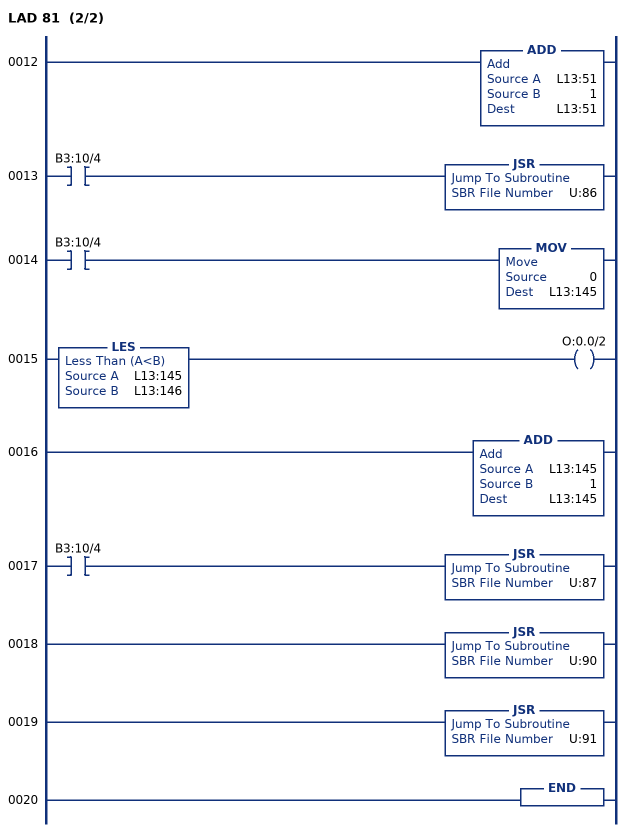
% Rung: 12 %
SOR ADD L13:51 1 L13:51 EOR
% Rung: 13 %
SOR XIC B3:10/4 JSR U:86 EOR
% Rung: 14 %
SOR XIC B3:10/4 MOV 0 L13:145 EOR
% Rung: 15 %
SOR LES L13:145 L13:146 OTE O:0.0/2 EOR
% Rung: 16 %
SOR ADD L13:145 1 L13:145 EOR
% Rung: 17 %
SOR XIC B3:10/4 JSR U:87 EOR
% Rung: 18 %
SOR JSR U:90 EOR
% Rung: 19 %
SOR JSR U:91 EOR
% Rung: 20 %
SOR END EOR

LADDER 82
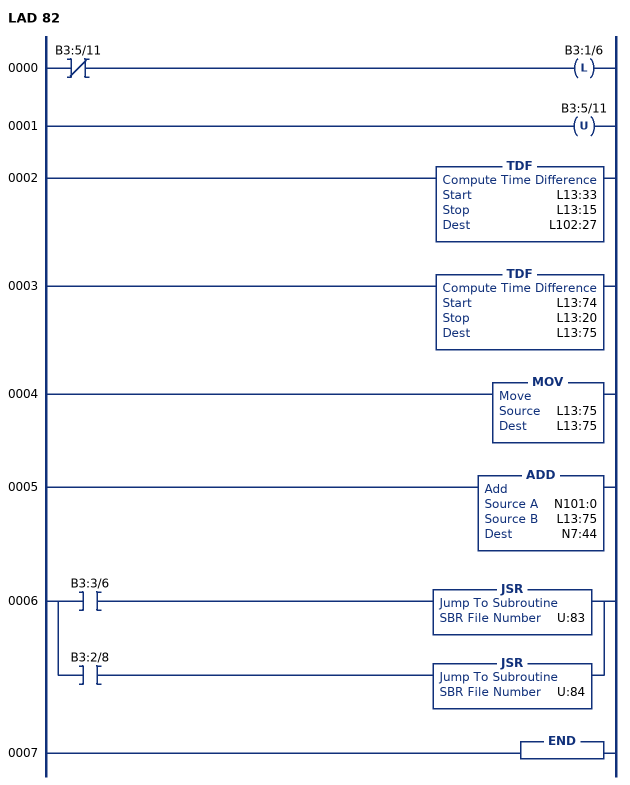
% Rung: 0 %
SOR XIO B3:5/11 OTL B3:1/6 EOR
% Rung: 1 %
SOR OTU B3:5/11 EOR
% Rung: 2 %
SOR TDF L13:33 L13:15 L102:27 EOR
% Rung: 3 %
SOR TDF L13:74 L13:20 L13:75 EOR
% Rung: 4 %
SOR MOV L13:75 L13:75 EOR
% Rung: 5 %
SOR ADD N101:0 L13:75 N7:44 EOR
% Rung: 6 %
SOR BST XIC B3:3/6 JSR U:83 NXB XIC B3:2/8 JSR U:84 BND EOR
% Rung: 7 %
SOR END EOR

LADDER 83
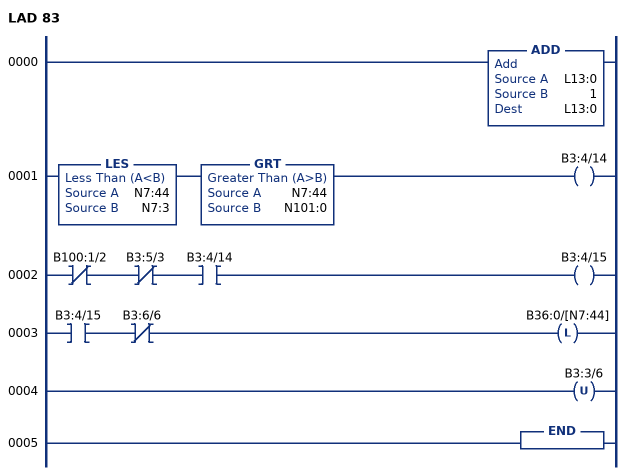
% Rung: 0 %
SOR ADD L13:0 1 L13:0 EOR
% Rung: 1 %
SOR LES N7:44 N7:3 GRT N7:44 N101:0 OTE B3:4/14 EOR
% Rung: 2 %
SOR XIO B100:1/2 XIO B3:5/3 XIC B3:4/14 OTE B3:4/15 EOR
% Rung: 3 %
SOR XIC B3:4/15 XIO B3:6/6 OTL B36:0/[N7:44] EOR
% Rung: 4 %
SOR OTU B3:3/6 EOR
% Rung: 5 %
SOR END EOR

LADDER 84
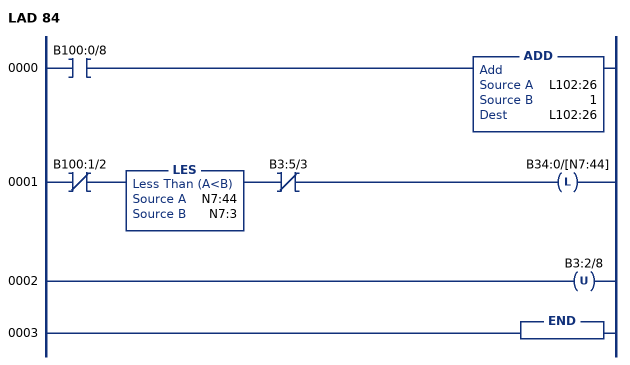
% Rung: 0 %
SOR XIC B100:0/8 ADD L102:26 1 L102:26 EOR
% Rung: 1 %
SOR XIO B100:1/2 LES N7:44 N7:3 XIO B3:5/3 OTL B34:0/[N7:44] EOR
% Rung: 2 %
SOR OTU B3:2/8 EOR
% Rung: 3 %
SOR END EOR

LADDER 85
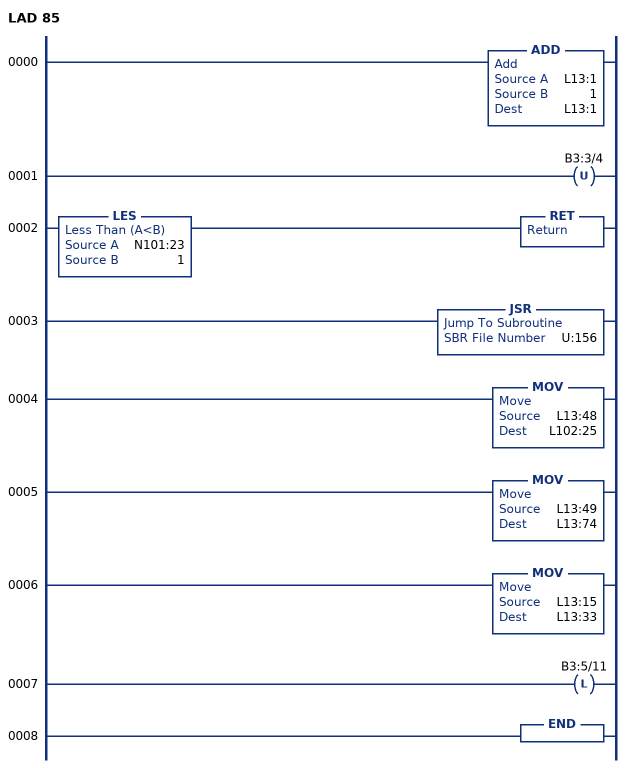
% Rung: 0 %
SOR ADD L13:1 1 L13:1 EOR
% Rung: 1 %
SOR OTU B3:3/4 EOR
% Rung: 2 %
SOR LES N101:23 1 RET EOR
% Rung: 3 %
SOR JSR U:156 EOR
% Rung: 4 %
SOR MOV L13:48 L102:25 EOR
% Rung: 5 %
SOR MOV L13:49 L13:74 EOR
% Rung: 6 %
SOR MOV L13:15 L13:33 EOR
% Rung: 7 %
SOR OTL B3:5/11 EOR
% Rung: 8 %
SOR END EOR

LADDER 86
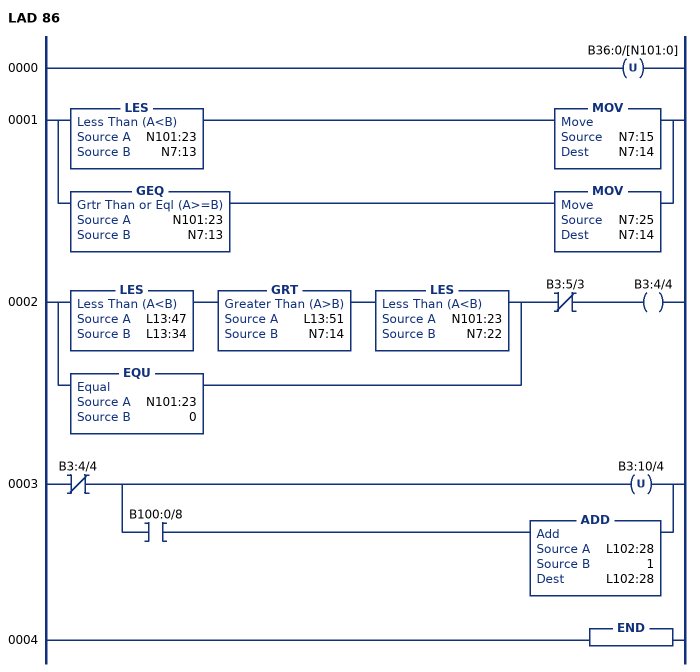
% Rung: 0 %
SOR OTU B36:0/[N101:0] EOR
% Rung: 1 %
SOR BST LES N101:23 N7:13 MOV N7:15 N7:14 NXB GEQ N101:23 N7:13 MOV N7:25 N7:14 BND EOR
% Rung: 2 %
SOR BST LES L13:47 L13:34 GRT L13:51 N7:14 LES N101:23 N7:22 NXB EQU N101:23 0 BND XIO B3:5/3 OTE B3:4/4 EOR
% Rung: 3 %
SOR XIO B3:4/4 BST OTU B3:10/4 NXB XIC B100:0/8 ADD L102:28 1 L102:28 BND EOR
% Rung: 4 %
SOR END EOR

LADDER 87
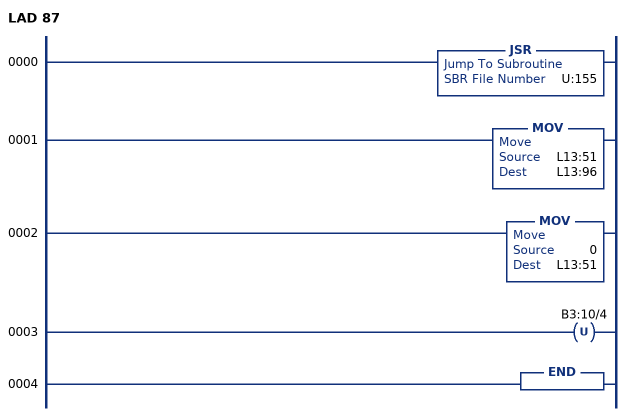
% Rung: 0 %
SOR JSR U:155 EOR
% Rung: 1 %
SOR MOV L13:51 L13:96 EOR
% Rung: 2 %
SOR MOV 0 L13:51 EOR
% Rung: 3 %
SOR OTU B3:10/4 EOR
% Rung: 4 %
SOR END EOR

LADDER 90
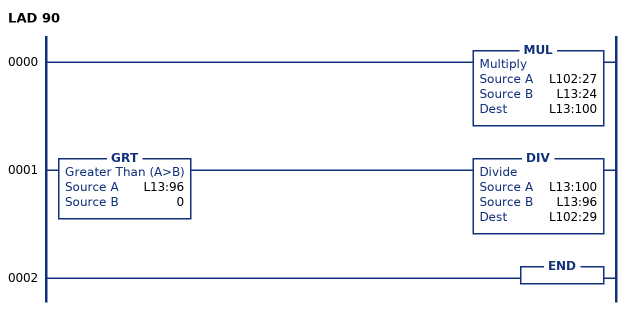
% Rung: 0 %
SOR MUL L102:27 L13:24 L13:100 EOR
% Rung: 1 %
SOR GRT L13:96 0 DIV L13:100 L13:96 L102:29 EOR
% Rung: 2 %
SOR END EOR

LADDER 91
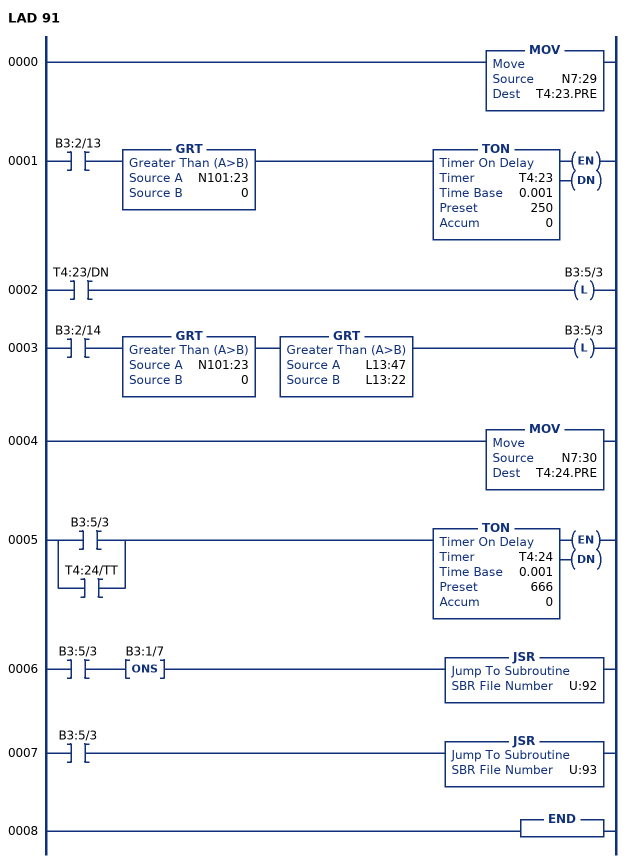
% Rung: 0 %
SOR MOV N7:29 T4:23.PRE EOR
% Rung: 1 %
SOR XIC B3:2/13 GRT N101:23 0 TON T4:23 0.001 250 0 EOR
% Rung: 2 %
SOR XIC T4:23/DN OTL B3:5/3 EOR
% Rung: 3 %
SOR XIC B3:2/14 GRT N101:23 0 GRT L13:47 L13:22 OTL B3:5/3 EOR
% Rung: 4 %
SOR MOV N7:30 T4:24.PRE EOR
% Rung: 5 %
SOR BST XIC B3:5/3 NXB XIC T4:24/TT BND TON T4:24 0.001 666 0 EOR
% Rung: 6 %
SOR XIC B3:5/3 ONS B3:1/7 JSR U:92 EOR
% Rung: 7 %
SOR XIC B3:5/3 JSR U:93 EOR
% Rung: 8 %
SOR END EOR

LADDER 92
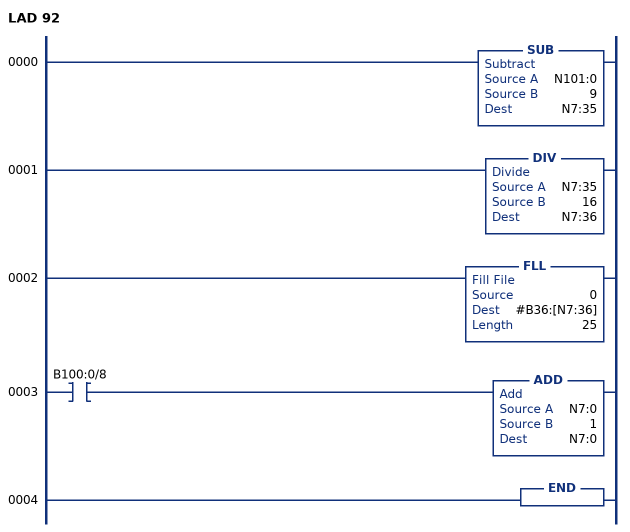
% Rung: 0 %
SOR SUB N101:0 9 N7:35 EOR
% Rung: 1 %
SOR DIV N7:35 16 N7:36 EOR
% Rung: 2 %
SOR FLL 0 #B36:[N7:36] 25 EOR
% Rung: 3 %
SOR XIC B100:0/8 ADD N7:0 1 N7:0 EOR
% Rung: 4 %
SOR END EOR

LADDER 93
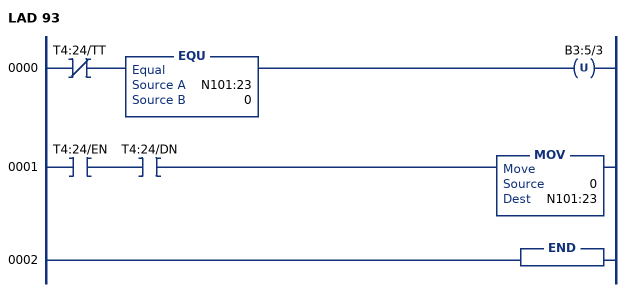
% Rung: 0 %
SOR XIO T4:24/TT EQU N101:23 0 OTU B3:5/3 EOR
% Rung: 1 %
SOR XIC T4:24/EN XIC T4:24/DN MOV 0 N101:23 EOR
% Rung: 2 %
SOR END EOR

LADDER 135
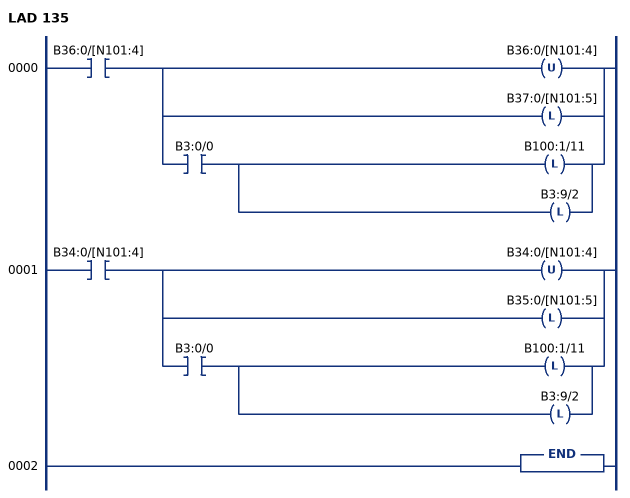
% Rung: 0 %
SOR XIC B36:0/[N101:4] BST OTU B36:0/[N101:4] NXB OTL B37:0/[N101:5] NXB XIC B3:0/0 BST OTL B100:1/11 NXB OTL B3:9/2 BND BND EOR
% Rung: 1 %
SOR XIC B34:0/[N101:4] BST OTU B34:0/[N101:4] NXB OTL B35:0/[N101:5] NXB XIC B3:0/0 BST OTL B100:1/11 NXB OTL B3:9/2 BND BND EOR
% Rung: 2 %
SOR END EOR

LADDER 137
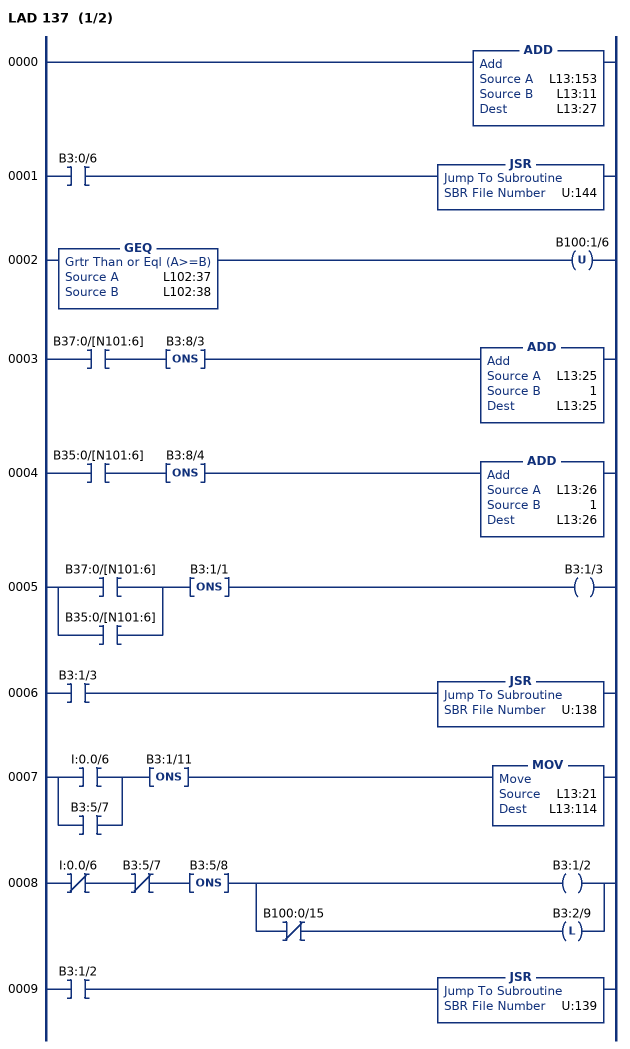
% Rung: 0 %
SOR ADD L13:153 L13:11 L13:27 EOR
% Rung: 1 %
SOR XIC B3:0/6 JSR U:144 EOR
% Rung: 2 %
SOR GEQ L102:37 L102:38 OTU B100:1/6 EOR
% Rung: 3 %
SOR XIC B37:0/[N101:6] ONS B3:8/3 ADD L13:25 1 L13:25 EOR
% Rung: 4 %
SOR XIC B35:0/[N101:6] ONS B3:8/4 ADD L13:26 1 L13:26 EOR
% Rung: 5 %
SOR BST XIC B37:0/[N101:6] NXB XIC B35:0/[N101:6] BND ONS B3:1/1 OTE B3:1/3 EOR
% Rung: 6 %
SOR XIC B3:1/3 JSR U:138 EOR
% Rung: 7 %
SOR BST XIC I:0.0/6 NXB XIC B3:5/7 BND ONS B3:1/11 MOV L13:21 L13:114 EOR
% Rung: 8 %
SOR XIO I:0.0/6 XIO B3:5/7 ONS B3:5/8 BST OTE B3:1/2 NXB XIO B100:0/15 OTL B3:2/9 BND EOR
% Rung: 9 %
SOR XIC B3:1/2 JSR U:139 EOR

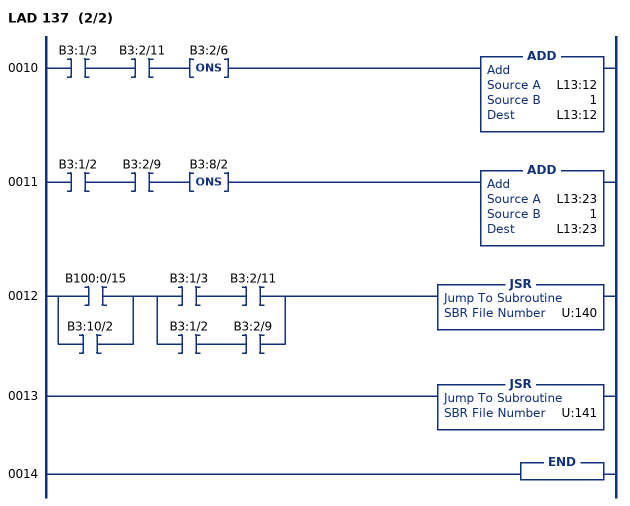
% Rung: 10 %
SOR XIC B3:1/3 XIC B3:2/11 ONS B3:2/6 ADD L13:12 1 L13:12 EOR
% Rung: 11 %
SOR XIC B3:1/2 XIC B3:2/9 ONS B3:8/2 ADD L13:23 1 L13:23 EOR
% Rung: 12 %
SOR BST XIC B100:0/15 NXB XIC B3:10/2 BND BST XIC B3:1/3 XIC B3:2/11 NXB XIC B3:1/2 XIC B3:2/9 BND JSR U:140 EOR
% Rung: 13 %
SOR JSR U:141 EOR
% Rung: 14 %
SOR END EOR

LADDER 138
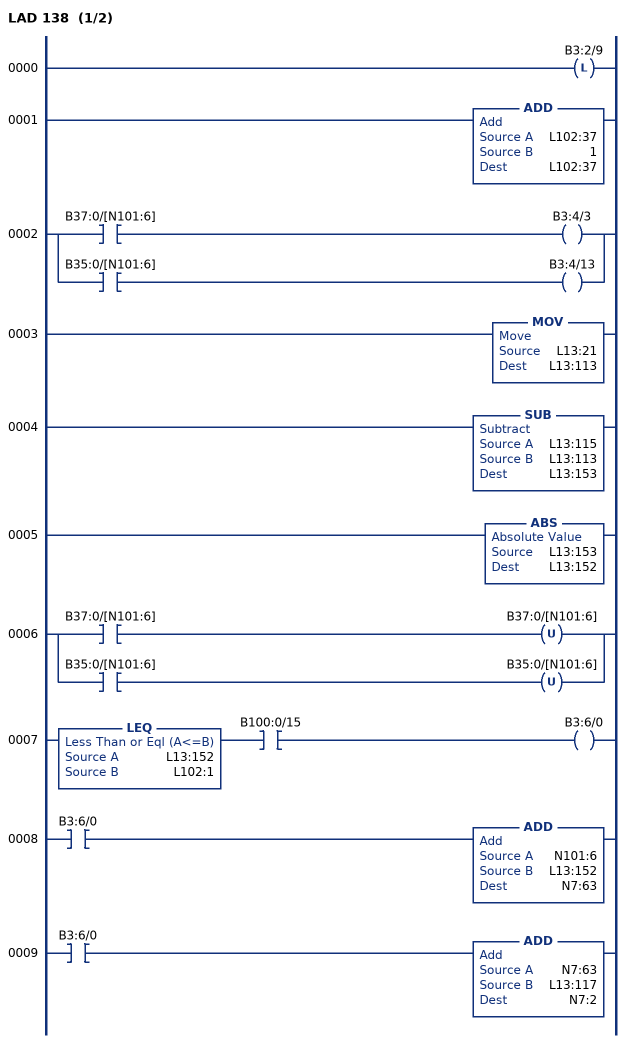
% Rung: 0 %
SOR OTL B3:2/9 EOR
% Rung: 1 %
SOR ADD L102:37 1 L102:37 EOR
% Rung: 2 %
SOR BST XIC B37:0/[N101:6] OTE B3:4/3 NXB XIC B35:0/[N101:6] OTE B3:4/13 BND EOR
% Rung: 3 %
SOR MOV L13:21 L13:113 EOR
% Rung: 4 %
SOR SUB L13:115 L13:113 L13:153 EOR
% Rung: 5 %
SOR ABS L13:153 L13:152 EOR
% Rung: 6 %
SOR BST XIC B37:0/[N101:6] OTU B37:0/[N101:6] NXB XIC B35:0/[N101:6] OTU B35:0/[N101:6] BND EOR
% Rung: 7 %
SOR LEQ L13:152 L102:1 XIC B100:0/15 OTE B3:6/0 EOR
% Rung: 8 %
SOR XIC B3:6/0 ADD N101:6 L13:152 N7:63 EOR
% Rung: 9 %
SOR XIC B3:6/0 ADD N7:63 L13:117 N7:2 EOR

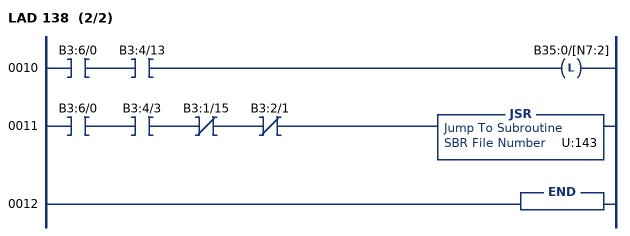
% Rung: 10 %
SOR XIC B3:6/0 XIC B3:4/13 OTL B35:0/[N7:2] EOR
% Rung: 11 %
SOR XIC B3:6/0 XIC B3:4/3 XIO B3:1/15 XIO B3:2/1 JSR U:143 EOR
% Rung: 12 %
SOR END EOR

LADDER 139
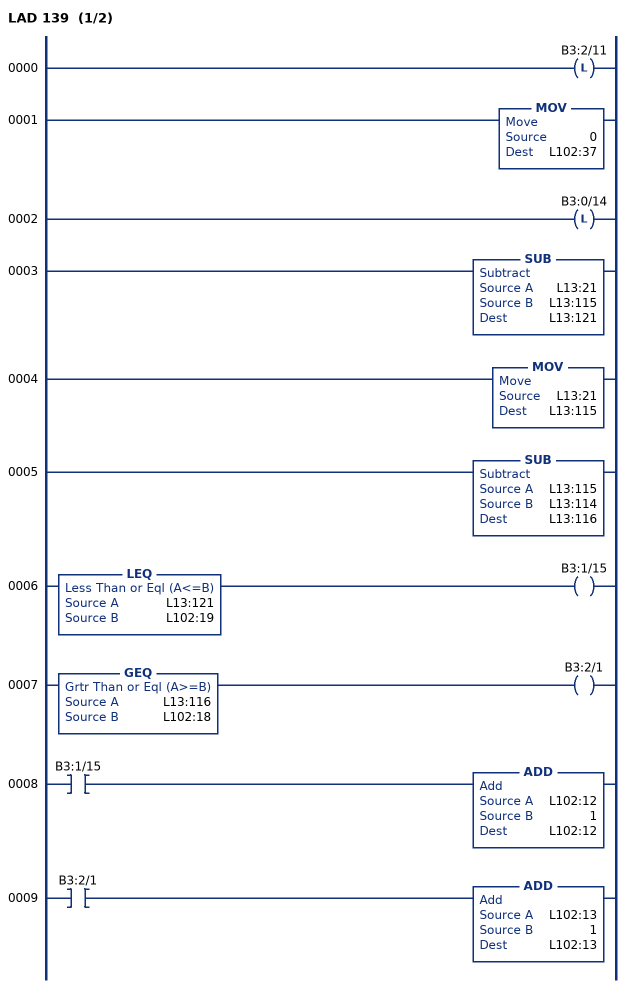
% Rung: 0 %
SOR OTL B3:2/11 EOR
% Rung: 1 %
SOR MOV 0 L102:37 EOR
% Rung: 2 %
SOR OTL B3:0/14 EOR
% Rung: 3 %
SOR SUB L13:21 L13:115 L13:121 EOR
% Rung: 4 %
SOR MOV L13:21 L13:115 EOR
% Rung: 5 %
SOR SUB L13:115 L13:114 L13:116 EOR
% Rung: 6 %
SOR LEQ L13:121 L102:19 OTE B3:1/15 EOR
% Rung: 7 %
SOR GEQ L13:116 L102:18 OTE B3:2/1 EOR
% Rung: 8 %
SOR XIC B3:1/15 ADD L102:12 1 L102:12 EOR
% Rung: 9 %
SOR XIC B3:2/1 ADD L102:13 1 L102:13 EOR

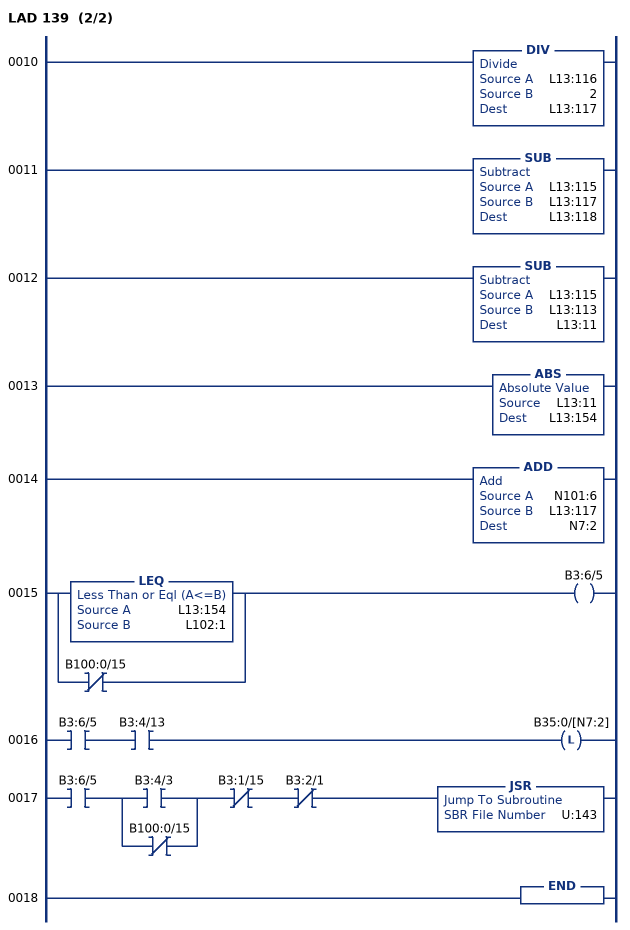
% Rung: 10 %
SOR DIV L13:116 2 L13:117 EOR
% Rung: 11 %
SOR SUB L13:115 L13:117 L13:118 EOR
% Rung: 12 %
SOR SUB L13:115 L13:113 L13:11 EOR
% Rung: 13 %
SOR ABS L13:11 L13:154 EOR
% Rung: 14 %
SOR ADD N101:6 L13:117 N7:2 EOR
% Rung: 15 %
SOR BST LEQ L13:154 L102:1 NXB XIO B100:0/15 BND OTE B3:6/5 EOR
% Rung: 16 %
SOR XIC B3:6/5 XIC B3:4/13 OTL B35:0/[N7:2] EOR
% Rung: 17 %
SOR XIC B3:6/5 BST XIC B3:4/3 NXB XIO B100:0/15 BND XIO B3:1/15 XIO B3:2/1 JSR U:143 EOR
% Rung: 18 %
SOR END EOR

LADDER 140
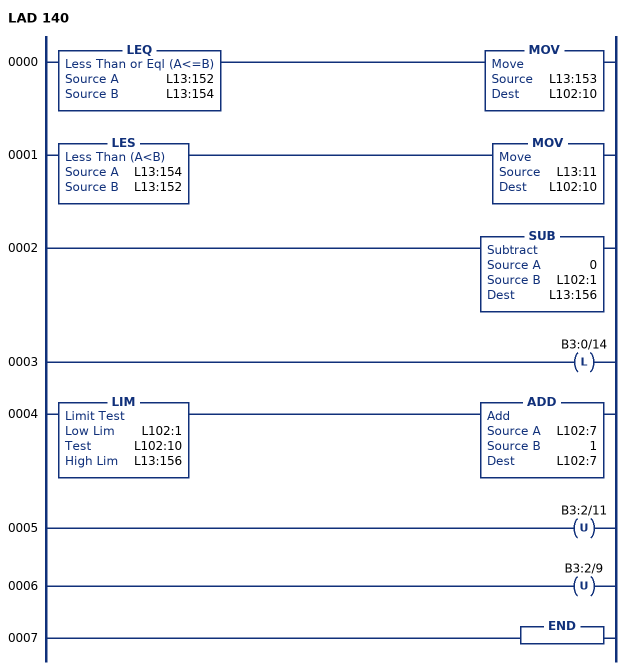
% Rung: 0 %
SOR LEQ L13:152 L13:154 MOV L13:153 L102:10 EOR
% Rung: 1 %
SOR LES L13:154 L13:152 MOV L13:11 L102:10 EOR
% Rung: 2 %
SOR SUB 0 L102:1 L13:156 EOR
% Rung: 3 %
SOR OTL B3:0/14 EOR
% Rung: 4 %
SOR LIM L102:1 L102:10 L13:156 ADD L102:7 1 L102:7 EOR
% Rung: 5 %
SOR OTU B3:2/11 EOR
% Rung: 6 %
SOR OTU B3:2/9 EOR
% Rung: 7 %
SOR END EOR

LADDER 141
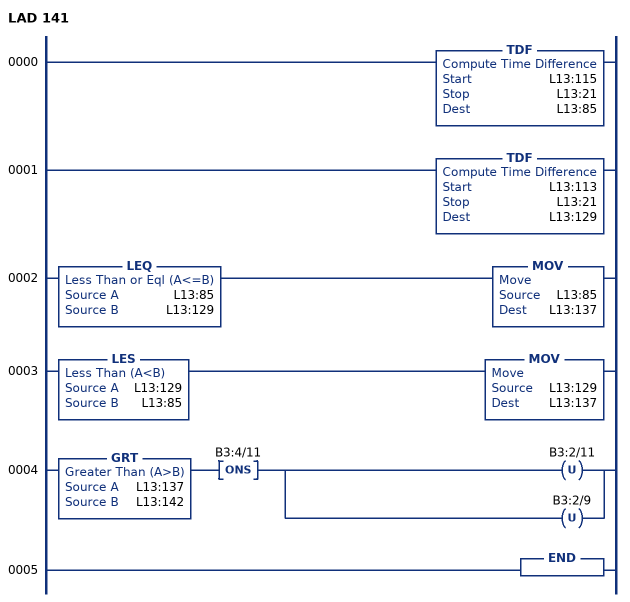
% Rung: 0 %
SOR TDF L13:115 L13:21 L13:85 EOR
% Rung: 1 %
SOR TDF L13:113 L13:21 L13:129 EOR
% Rung: 2 %
SOR LEQ L13:85 L13:129 MOV L13:85 L13:137 EOR
% Rung: 3 %
SOR LES L13:129 L13:85 MOV L13:129 L13:137 EOR
% Rung: 4 %
SOR GRT L13:137 L13:142 ONS B3:4/11 BST OTU B3:2/11 NXB OTU B3:2/9 BND EOR
% Rung: 5 %
SOR END EOR

LADDER 142
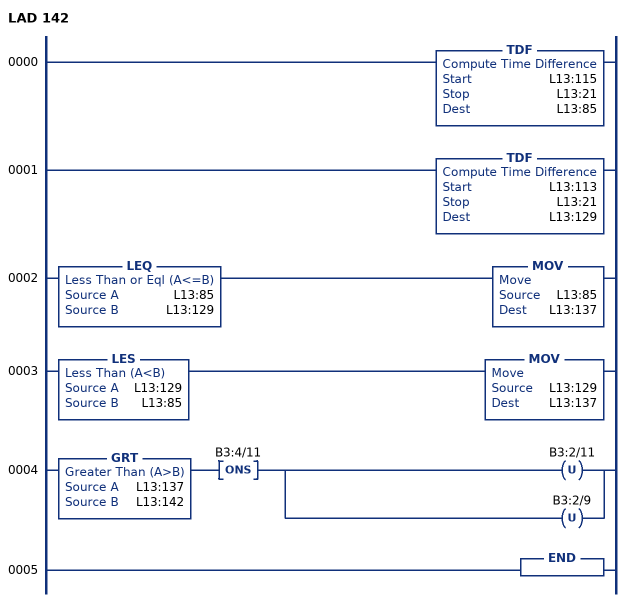
% Rung: 0 %
SOR TDF L13:115 L13:21 L13:85 EOR
% Rung: 1 %
SOR TDF L13:113 L13:21 L13:129 EOR
% Rung: 2 %
SOR LEQ L13:85 L13:129 MOV L13:85 L13:137 EOR
% Rung: 3 %
SOR LES L13:129 L13:85 MOV L13:129 L13:137 EOR
% Rung: 4 %
SOR GRT L13:137 L13:142 ONS B3:4/11 BST OTU B3:2/11 NXB OTU B3:2/9 BND EOR
% Rung: 5 %
SOR END EOR

LADDER 143
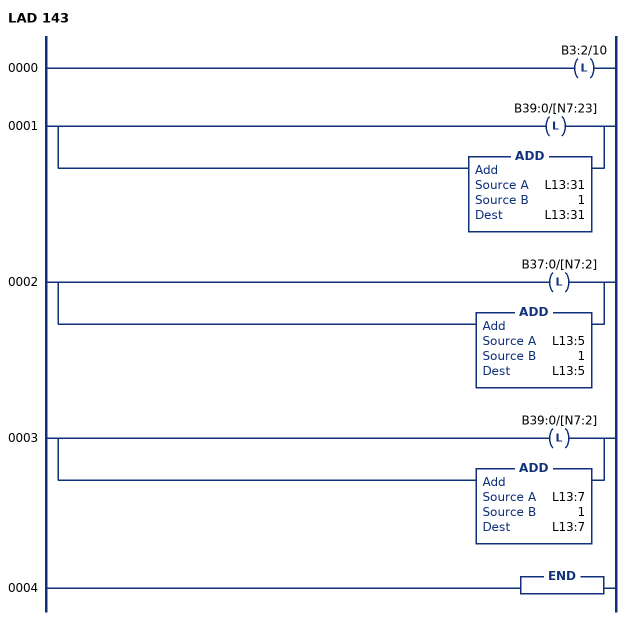
% Rung: 0 %
SOR OTL B3:2/10 EOR
% Rung: 1 %
SOR BST OTL B39:0/[N7:23] NXB ADD L13:31 1 L13:31 BND EOR
% Rung: 2 %
SOR BST OTL B37:0/[N7:2] NXB ADD L13:5 1 L13:5 BND EOR
% Rung: 3 %
SOR BST OTL B39:0/[N7:2] NXB ADD L13:7 1 L13:7 BND EOR
% Rung: 4 %
SOR END EOR

LADDER 144
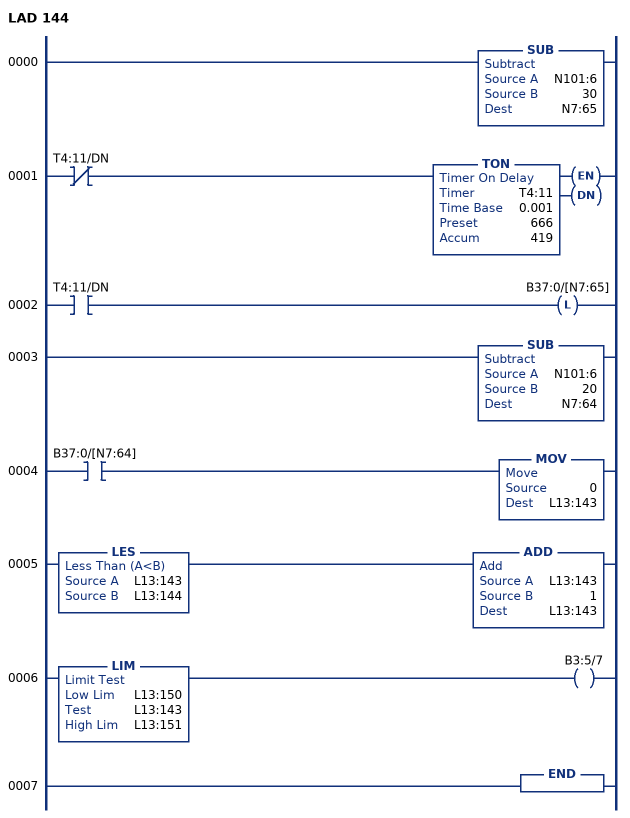
% Rung: 0 %
SOR SUB N101:6 30 N7:65 EOR
% Rung: 1 %
SOR XIO T4:11/DN TON T4:11 0.001 666 419 EOR
% Rung: 2 %
SOR XIC T4:11/DN OTL B37:0/[N7:65] EOR
% Rung: 3 %
SOR SUB N101:6 20 N7:64 EOR
% Rung: 4 %
SOR XIC B37:0/[N7:64] MOV 0 L13:143 EOR
% Rung: 5 %
SOR LES L13:143 L13:144 ADD L13:143 1 L13:143 EOR
% Rung: 6 %
SOR LIM L13:150 L13:143 L13:151 OTE B3:5/7 EOR
% Rung: 7 %
SOR END EOR

LADDER 148
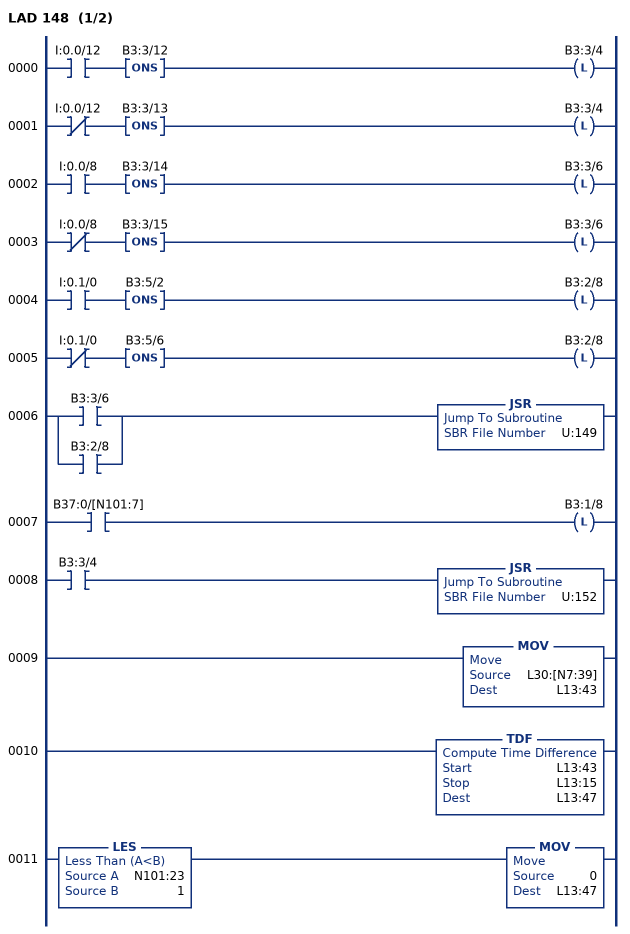
% Rung: 0 %
SOR XIC I:0.0/12 ONS B3:3/12 OTL B3:3/4 EOR
% Rung: 1 %
SOR XIO I:0.0/12 ONS B3:3/13 OTL B3:3/4 EOR
% Rung: 2 %
SOR XIC I:0.0/8 ONS B3:3/14 OTL B3:3/6 EOR
% Rung: 3 %
SOR XIO I:0.0/8 ONS B3:3/15 OTL B3:3/6 EOR
% Rung: 4 %
SOR XIC I:0.1/0 ONS B3:5/2 OTL B3:2/8 EOR
% Rung: 5 %
SOR XIO I:0.1/0 ONS B3:5/6 OTL B3:2/8 EOR
% Rung: 6 %
SOR BST XIC B3:3/6 NXB XIC B3:2/8 BND JSR U:149 EOR
% Rung: 7 %
SOR XIC B37:0/[N101:7] OTL B3:1/8 EOR
% Rung: 8 %
SOR XIC B3:3/4 JSR U:152 EOR
% Rung: 9 %
SOR MOV L30:[N7:39] L13:43 EOR
% Rung: 10 %
SOR TDF L13:43 L13:15 L13:47 EOR
% Rung: 11 %
SOR LES N101:23 1 MOV 0 L13:47 EOR

